TYPE ST_Listentry :
STRUCT
	nRawId		: INT;
	nId			: INT;
	bEnable		: BOOL;
	sName		: STRING;
END_STRUCT
END_TYPE

(* stored: Version 1.1.0.1
   DUT ST_Listentry: Id {4d62ebaf-c98c-475b-8e15-f14fdd584cf7} *)
